{attribute addProperty BoxType "EL4038-0000-0018"}
{attribute addProperty Id "AO_Output_ChannelAT %Q*ARRAY[0..7] OF AO_Output_Channel_F57FA4F9128160WcStateAT %I*WcState_28A8677510.1250InfoDataAT %I*InfoData_BC63D37F80100"}
{attribute addProperty CRC "3986678857"}
{attribute addProperty SizeInBites "209"}
{attribute addProperty SizeInBytes "26.125"}
TYPE EL4038_5F89906A :
STRUCT
	{attribute addProperty Name "AO_Output_Channel"}
	AO_Output_Channel : ARRAY[0..7] OF AO_Output_Channel_F57FA4F9;
	{attribute addProperty Name "WcState"}
	WcState : WcState_28A86775;
	{attribute addProperty Name "InfoData"}
	InfoData : InfoData_BC63D37F;
END_STRUCT
END_TYPE

(* stored: Version 1.2.0.0, ProductVersion 3.1.4024.9
   DUT EL4038_5F89906A: Id {926042ec-263f-4c59-8663-2c33de129277} *)
